Fanuc KAREL source: kd00046.KL

-- PROVISIONAL review KL for V1013-1; original PC SHA256 410eae32a4926c5ea0af5ed57547aa60c14f6d42905ba7d45341e659ce611e50
-- Incomplete behavior may be omitted. Consult companion uncertainty JSON. Do not deploy.
PROGRAM KD00046
%NOLOCKGROUP
VAR
  I : INTEGER
  J : INTEGER
  B : BOOLEAN
  R : REAL
  S : STRING[80]
-- UNRESOLVED_DECL V type=000013
BEGIN
  -- UNRESOLVED_PC offsets 5-20; opcodes 2E,22,32,35
  -- UNRESOLVED_PC offsets 25-41; opcodes 01,49,0A,82,0B
  -- UNRESOLVED_PC offsets 46-50; opcodes 7F
END KD00046
